// TIA Portal project "Analog İşlemler" (V17)

(* hardware
DEVICE "S7-1200 station_1"  S7-1200 Station
   slot 0: "Rack_0"  S7-1200 Rack  Rack  V1.0
   slot 1: "PLC_1"  CPU 1212C AC/DC/Rly  6ES7 212-1BE40-0XB0  V4.4
*)

// ===== PLC "PLC_1"  CPU 1212C AC/DC/Rly =====

VAR_GLOBAL   // PLC tag table "Default tag table"
   "Tag_1" AT %I0.0 : Bool;
   "Tag_2" AT %Q0.0 : Bool;
   "System_Byte" AT %MB20 : Byte;
   "FirstScan" AT %M20.0 : Bool;
   "DiagStatusUpdate" AT %M20.1 : Bool;
   "AlwaysTRUE" AT %M20.2 : Bool;
   "AlwaysFALSE" AT %M20.3 : Bool;
   "Clock_Byte" AT %MB25 : Byte;
   "Clock_10Hz" AT %M25.0 : Bool;
   "Clock_5Hz" AT %M25.1 : Bool;
   "Clock_2.5Hz" AT %M25.2 : Bool;
   "Clock_2Hz" AT %M25.3 : Bool;
   "Clock_1.25Hz" AT %M25.4 : Bool;
   "Clock_1Hz" AT %M25.5 : Bool;
   "Clock_0.625Hz" AT %M25.6 : Bool;
   "Clock_0.5Hz" AT %M25.7 : Bool;
   "Tag_3" AT %I0.1 : Bool;
   "Tag_4" AT %QB0 : Byte;
   "Tag_5" AT %I0.2 : Bool;
   "Tag_6" AT %MB2 : Byte;
   "Tag_7" AT %M100.0 : Bool;
   "Tag_8" AT %MW0 : Int;
   "Tag_9" AT %Q0.1 : Bool;
   "Tag_10" AT %Q0.2 : Bool;
   "Tag_11" AT %IW64 : Word;
   "Tag_12" AT %MW10 : Word;
   "Tag_13" AT %MD10 : Real;
END_VAR

ORGANIZATION_BLOCK "Main"   // OB1, LAD, ProgramCycle
TITLE = "Main Program Sweep (Cycle)"
{ S7_Optimized_Access := 'TRUE' }
VERSION : 0.1
   VAR_INPUT
      Initial_Call : Bool;   // Initial call of this OB
      Remanence : Bool;   // =True, if remanent data are available
   END_VAR
BEGIN

REGION Network 1
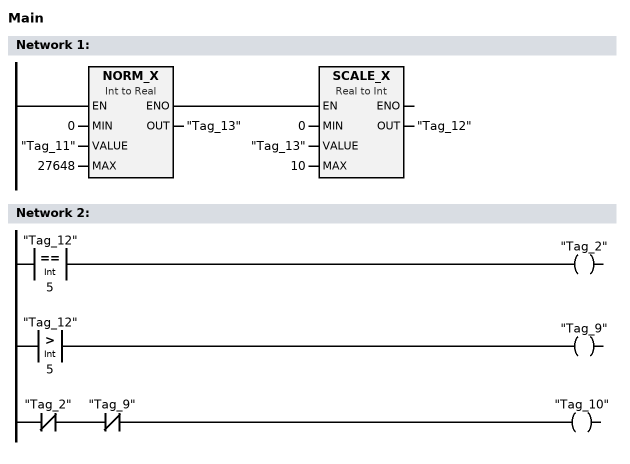
   RUNG wire#powerrail
      { S7_Templates := "[SrcType := Int, DestType := Real]" } Normalize(min := 0, value := "Tag_11", max := 27648, out => "Tag_13")
      { S7_Templates := "[SrcType := Real, DestType := Int]" } Scale(min := 0, value := "Tag_13", max := 10, out => "Tag_12")
   END_RUNG
   // the same network as SCL:
   "Tag_13" := NORM_X(MIN := 0, VALUE := "Tag_11", MAX := 27648);
   "Tag_12" := SCALE_X(MIN := 0, VALUE := "Tag_13", MAX := 10);
END_REGION

REGION Network 2
   RUNG wire#powerrail
      { S7_Templates := "SrcType := Int" } EQ_Contact(in1 := "Tag_12", in2 := 5)
      Coil( "Tag_2" )
   END_RUNG
   RUNG wire#powerrail
      { S7_Templates := "SrcType := Int" } GT_Contact(in1 := "Tag_12", in2 := 5)
      Coil( "Tag_9" )
   END_RUNG
   RUNG wire#powerrail
      I_Contact( "Tag_2" )
      I_Contact( "Tag_9" )
      Coil( "Tag_10" )
   END_RUNG
   // the same network as SCL:
   "Tag_2" := "Tag_12" = 5;
   "Tag_9" := "Tag_12" > 5;
   "Tag_10" := NOT "Tag_2" AND NOT "Tag_9";
END_REGION
END_ORGANIZATION_BLOCK